TYPE ST_AxisIn :
STRUCT
	/// Ec Box State
	iEcState				: UINT;
	/// Motortemp: [1/10 °C]
	iMotorTemperature		: INT;
	/// Amplifiertemp: [1/10 °C]
	iAmplifierTemperature	: INT;
	/// Versorgungsspannung
	iActualMainVoltage		: INT;
	/// User Status Wort
	nUserStateWord			: WORD;
END_STRUCT
END_TYPE

(* stored: Version 1.1.0.1, ProductVersion 3.1.4024.12
   DUT ST_AxisIn: Id {38e87050-7532-475a-a3f1-0a199d211c58} *)
